(* IEC 61131-3 sources: plcassist-cli/packages/volt-lsp-iec/test-corpus/twincat-project14/POUs, 3 files *)

(* ---- VltFixtureCfc.fb ---- *)
FUNCTION_BLOCK VltFixtureCfc
VAR_INPUT
END_VAR
VAR_OUTPUT
END_VAR
VAR
END_VAR

(* @volt-graphical: CFC *)

END_FUNCTION_BLOCK

(* ---- VltFixtureSfc.fb ---- *)
FUNCTION_BLOCK VltFixtureSfc
VAR_INPUT
END_VAR
VAR_OUTPUT
END_VAR
VAR
END_VAR

(* @volt-graphical: SFC *)

END_FUNCTION_BLOCK

(* ---- POUexecute.prg ---- *)
PROGRAM POUexecute
VAR
	iCount:INT;

	t1: TON;
	output: BOOL;
	e1: TIME;
	in1: BOOL;
	a: BOOL;
	b: BOOL;
	c: BOOL;
	out1: BOOL;
	t2: TON;
	out2: INT;
END_VAR

NETWORK 0 LD
  LET en1 := TRUE;
  IF en1 THEN
  EXECUTE
iCount:=icount+1;
  END_EXECUTE
  END_IF
END_NETWORK
NETWORK 1 LD
  output := t1(IN := in1, PT := e1);
END_NETWORK
NETWORK 2 LD
  LET g1 := b;
  out1 := ((a OR g1) AND c);
  out2 := g1;
END_NETWORK
NETWORK 3 LD
  output := t2(IN := , PT := e1);
END_NETWORK

END_PROGRAM
